FUNCTION_BLOCK CustomDeserializationFailedError_TestSuite EXTENDS TcUnit.FB_TestSuite

TestAccept();
TestErrorType();
TestIsSameAsWithSameErrors();
TestIsSameAsWithDifferentErrors();
TestMessage();
TestSerializeWith();

METHOD PUBLIC TestAccept
VAR
	error : CustomDeserializationFailedError(Message := 'TestMessage');
	visitor : MockVisitor(ExpectedError := error);
END_VAR
TEST('TestAccept');

error.Accept(visitor);

AssertTrue(
	Condition := visitor.VisitedCorrectError,
	Message := 'Did not invoke VisitError on the visitor'
);

TEST_FINISHED();
END_METHOD

METHOD PUBLIC TestErrorType
VAR
	error : CustomDeserializationFailedError(Message := 'TestMessage');
END_VAR
TEST('TestErrorType');

AssertEquals_String(
	Actual := error.ErrorType,
	Expected := 'CUSTOM_DESERIALIZATION_ERROR',
	Message := 'Did not return the expected ErrorType'
);

TEST_FINISHED();
END_METHOD

METHOD PUBLIC TestIsSameAsWithDifferentErrors
VAR
	error1 : CustomDeserializationFailedError(Message := 'TestMessage');
	error2 : MockError(MockErrorType:='ERROR_TYPE_B',MockMessage:='TestMessage');
END_VAR
TEST('TestIsSameAsWithDifferentErrors');

AssertFalse(
	Condition := error1.IsSameAs(error2),
	Message := 'Did not correctly identify errors as being different type'
);

TEST_FINISHED();
END_METHOD

METHOD PUBLIC TestIsSameAsWithSameErrors
VAR
	error1 : CustomDeserializationFailedError(Message := 'TestMessage');
	error2 : MockError(MockErrorType:='CUSTOM_DESERIALIZATION_ERROR',MockMessage:='Deserialization Failed, TestMessage');
END_VAR
TEST('TestIsSameAsWithSameErrors');

AssertTrue(
	Condition := error1.IsSameAs(error2),
	Message := 'Did not correctly identify errors as being the same type'
);

TEST_FINISHED();
END_METHOD

METHOD PUBLIC TestMessage
VAR
	error : CustomDeserializationFailedError(Message := 'TestMessage');
END_VAR
TEST('TestMessage');

AssertEquals_String(
	Actual := error.Message,
	Expected := 'Deserialization Failed, TestMessage',
	Message := 'Did not return the expected Message'
);

TEST_FINISHED();
END_METHOD

METHOD PUBLIC TestSerializeWith
VAR
	error : CustomDeserializationFailedError(Message := 'TestMessage');
	serializer : MockJsonSerializer;
	result : T_MAXSTRING;
END_VAR
TEST('TestSerializeWith');

error.SerializeWith(serializer);
serializer.TryGetSerializedData(ADR(result), SIZEOF(result));

AssertEquals_String(
	Actual := result,
	Expected := '{"errorType":"CUSTOM_DESERIALIZATION_ERROR","message":"Deserialization Failed, TestMessage"}',
	Message := 'Did not serialize correctly'
);

TEST_FINISHED();
END_METHOD

END_FUNCTION_BLOCK

(* stored: Version 1.1.0.1, ProductVersion 3.1.4024.12
   POU CustomDeserializationFailedError_TestSuite: Id {fa0d09c9-b154-0b31-0a63-257a16fa47df}, SpecialFunc None
   Method TestAccept: Id {b82ebc90-7911-05cc-1974-29186f172e66}
   Method TestErrorType: Id {feb45d11-c836-03b1-1eb8-a468b3e8b683}
   Method TestIsSameAsWithDifferentErrors: Id {67b4b579-c80d-0e65-250d-db0104d15a79}
   Method TestIsSameAsWithSameErrors: Id {65009b05-0dc3-01fb-0713-2406322c93ad}
   Method TestMessage: Id {03270791-0cbe-07e1-254f-726467faf9f2}
   Method TestSerializeWith: Id {b0b825b2-943a-002a-2947-89fd7501af3a} *)
